(* CoDeSys 2.3.9.37 project: CapB_3.pro *)
(* Libraries: Standard.lib 4.10.05 12:14:46 *)

(* POU PLC_PRG, ST *)
PROGRAM PLC_PRG
VAR
  Alarma:BOOL;
  Invisible: BOOL;
  Desactiva:BOOL;
	Numero: INT;
END_VAR
;
END_PROGRAM

(* Visualisation EjemploVisu
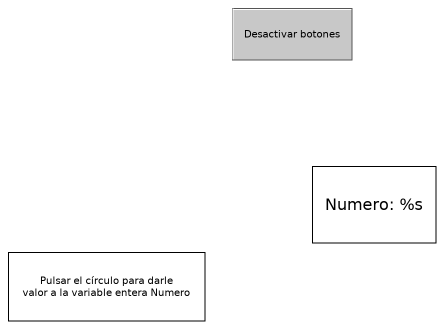
button at (249,36)-(369,88): text "Desactivar botones"; toggles PLC_PRG.Desactiva
rectangle at (25,280)-(222,349): text "Pulsar el círculo para darle / valor a la variable entera Numero"
rectangle at (329,194)-(453,271): text "Numero: %s"; shows PLC_PRG.Numero
3 elements of other kinds (tables, trends, ...) not read
*)
